PROGRAM ST5_MOTOR_1
VAR
	ClearFault: FB_ClearFault;
	SetEnableState: FB_SetEnableState;
	SetHomingParameter: FB_SetHomingParameter;
	FindHome: FB_FindHome;
	POSITION: DINT;
	GetMovementState: FB_GetMovementState;
	MoveToPosition: FB_MoveToPosition;
	SetOperationMode: FB_SetOperationMode;
	SetMotorParameter: FB_SetMotorParameter;
	SetPositionProfile: FB_SetPositionProfile;
END_VAR

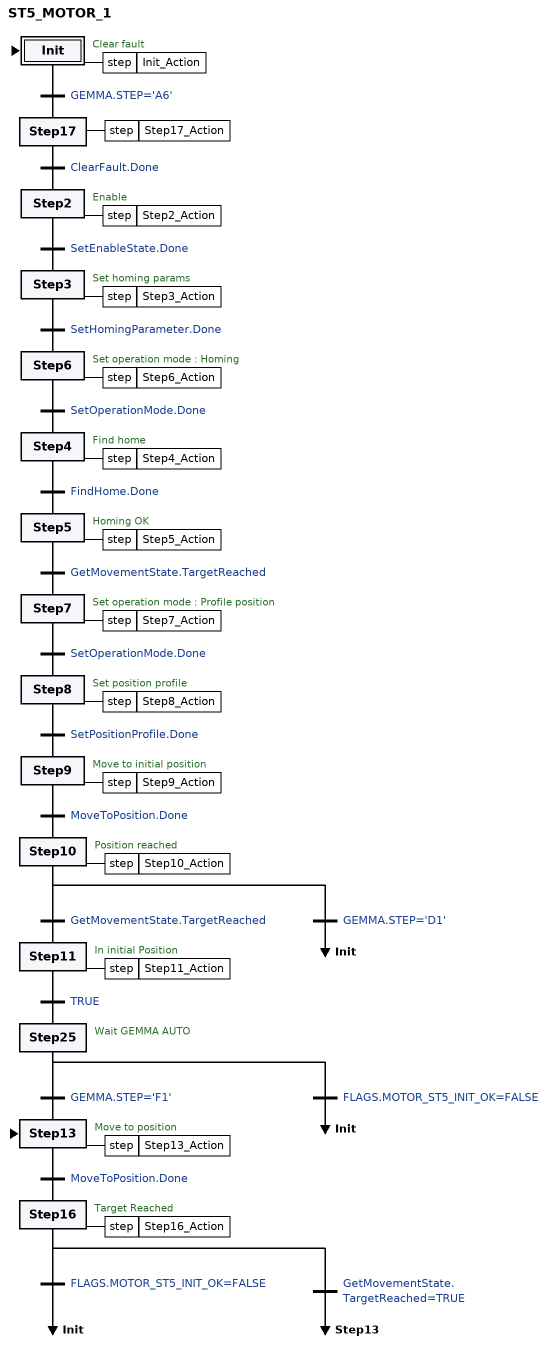
// Clear fault
INITIAL_STEP Init:
    Init_Action(N);  // step action
END_STEP
TRANSITION FROM Init TO Step17
    := GEMMA.STEP='A6';
END_TRANSITION
STEP Step17:
    Step17_Action(N);  // step action
END_STEP
TRANSITION FROM Step17 TO Step2
    := ClearFault.Done;
END_TRANSITION
// Enable
STEP Step2:
    Step2_Action(N);  // step action
END_STEP
TRANSITION FROM Step2 TO Step3
    := SetEnableState.Done;
END_TRANSITION
// Set homing params
STEP Step3:
    Step3_Action(N);  // step action
END_STEP
TRANSITION FROM Step3 TO Step6
    := SetHomingParameter.Done;
END_TRANSITION
// Set operation mode : Homing
STEP Step6:
    Step6_Action(N);  // step action
END_STEP
TRANSITION FROM Step6 TO Step4
    := SetOperationMode.Done;
END_TRANSITION
// Find home
STEP Step4:
    Step4_Action(N);  // step action
END_STEP
TRANSITION FROM Step4 TO Step5
    := FindHome.Done;
END_TRANSITION
// Homing OK
STEP Step5:
    Step5_Action(N);  // step action
END_STEP
TRANSITION FROM Step5 TO Step7
    := GetMovementState.TargetReached;
END_TRANSITION
// Set operation mode : Profile position
STEP Step7:
    Step7_Action(N);  // step action
END_STEP
TRANSITION FROM Step7 TO Step8
    := SetOperationMode.Done;
END_TRANSITION
// Set position profile
STEP Step8:
    Step8_Action(N);  // step action
END_STEP
TRANSITION FROM Step8 TO Step9
    := SetPositionProfile.Done;
END_TRANSITION
// Move to initial position
STEP Step9:
    Step9_Action(N);  // step action
END_STEP
TRANSITION FROM Step9 TO Step10
    := MoveToPosition.Done;
END_TRANSITION
// Position reached
STEP Step10:
    Step10_Action(N);  // step action
END_STEP
TRANSITION FROM Step10 TO Step11
    := GetMovementState.TargetReached;
END_TRANSITION
TRANSITION FROM Step10 TO Init
    := GEMMA.STEP='D1';
END_TRANSITION
// In initial Position
STEP Step11:
    Step11_Action(N);  // step action
END_STEP
TRANSITION FROM Step11 TO Step25
    := TRUE;
END_TRANSITION
// Wait GEMMA AUTO
STEP Step25:
END_STEP
TRANSITION FROM Step25 TO Step13
    := GEMMA.STEP='F1';
END_TRANSITION
TRANSITION FROM Step25 TO Init
    := FLAGS.MOTOR_ST5_INIT_OK=FALSE;
END_TRANSITION
// Move to position
STEP Step13:
    Step13_Action(N);  // step action
END_STEP
TRANSITION FROM Step13 TO Step16
    := MoveToPosition.Done;
END_TRANSITION
// Target Reached
STEP Step16:
    Step16_Action(N);  // step action
END_STEP
TRANSITION FROM Step16 TO Init
    := FLAGS.MOTOR_ST5_INIT_OK=FALSE;
END_TRANSITION
TRANSITION FROM Step16 TO Step13
    := GetMovementState.TargetReached=TRUE;
END_TRANSITION

ACTION Step6_Action:
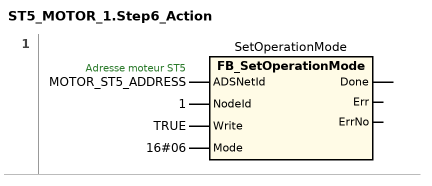
// NETWORK 1
//   MOTOR_ST5_ADDRESS: Adresse moteur ST5
SetOperationMode(ADSNetId := MOTOR_ST5_ADDRESS, NodeId := 1, Write := TRUE, Mode := 16#06); // FB_SetOperationMode
END_ACTION

ACTION Step2_Action:
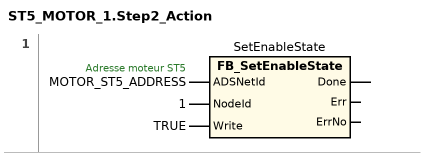
// NETWORK 1
//   MOTOR_ST5_ADDRESS: Adresse moteur ST5
SetEnableState(ADSNetId := MOTOR_ST5_ADDRESS, NodeId := 1, Write := TRUE); // FB_SetEnableState
END_ACTION

ACTION Step10_Action:
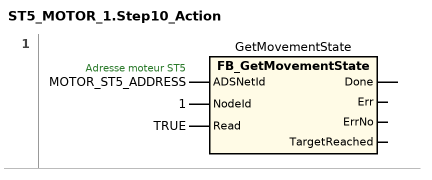
// NETWORK 1
//   MOTOR_ST5_ADDRESS: Adresse moteur ST5
GetMovementState(ADSNetId := MOTOR_ST5_ADDRESS, NodeId := 1, Read := TRUE); // FB_GetMovementState
END_ACTION

ACTION Step8_Action:
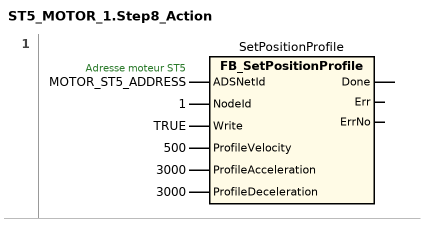
// NETWORK 1
//   MOTOR_ST5_ADDRESS: Adresse moteur ST5
SetPositionProfile(
    ADSNetId := MOTOR_ST5_ADDRESS,
    NodeId := 1,
    Write := TRUE,
    ProfileVelocity := 500,
    ProfileAcceleration := 3000,
    ProfileDeceleration := 3000); // FB_SetPositionProfile
END_ACTION

ACTION Step4_Action:
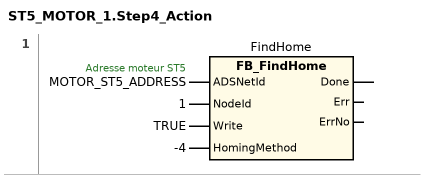
// NETWORK 1
//   MOTOR_ST5_ADDRESS: Adresse moteur ST5
FindHome(ADSNetId := MOTOR_ST5_ADDRESS, NodeId := 1, Write := TRUE, HomingMethod := -4); // FB_FindHome
END_ACTION

ACTION Step11_Action:

(*SetDisableState(
	ADSNetId:= '10.0.0.31.6.1',
	NodeId:= 1,
	Write:= TRUE);*)

FLAGS.MOTOR_ST5_INIT_OK:=TRUE;
END_ACTION

ACTION Step17_Action:
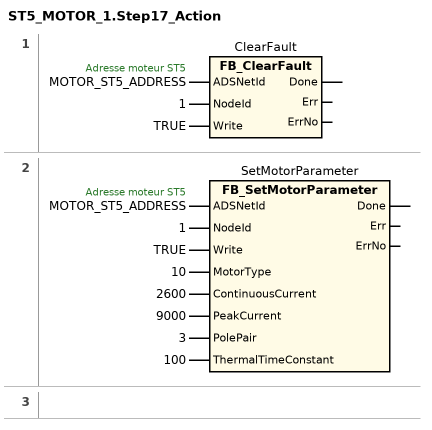
// NETWORK 1
//   MOTOR_ST5_ADDRESS: Adresse moteur ST5
ClearFault(ADSNetId := MOTOR_ST5_ADDRESS, NodeId := 1, Write := TRUE); // FB_ClearFault

// NETWORK 2
//   MOTOR_ST5_ADDRESS: Adresse moteur ST5
SetMotorParameter(
    ADSNetId := MOTOR_ST5_ADDRESS,
    NodeId := 1,
    Write := TRUE,
    MotorType := 10,
    ContinuousCurrent := 2600,
    PeakCurrent := 9000,
    PolePair := 3,
    ThermalTimeConstant := 100); // FB_SetMotorParameter

// NETWORK 3
END_ACTION

ACTION Step5_Action:
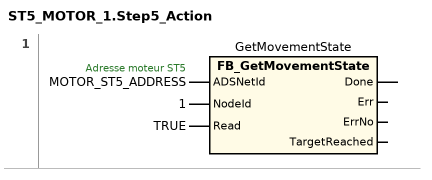
// NETWORK 1
//   MOTOR_ST5_ADDRESS: Adresse moteur ST5
GetMovementState(ADSNetId := MOTOR_ST5_ADDRESS, NodeId := 1, Read := TRUE); // FB_GetMovementState
END_ACTION

ACTION Step16_Action:
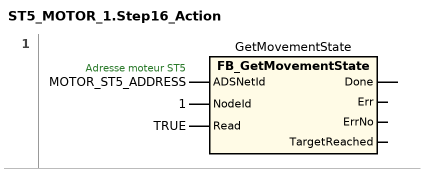
// NETWORK 1
//   MOTOR_ST5_ADDRESS: Adresse moteur ST5
GetMovementState(ADSNetId := MOTOR_ST5_ADDRESS, NodeId := 1, Read := TRUE); // FB_GetMovementState
END_ACTION

ACTION Init_Action:

END_ACTION

ACTION Step13_Action:
(*Limitation deplacement Moteur*)
IF FLAGS.MOTOR_ST5_POSITION>MOTOR_ST5_POSITION_MAX THEN
	POSITION:=MOTOR_ST5_POSITION_MAX;
ELSIF FLAGS.MOTOR_ST5_POSITION<0 THEN
	POSITION:=0;
ELSE
	POSITION:=FLAGS.MOTOR_ST5_POSITION;
END_IF


MoveToPosition(
	ADSNetId:= MOTOR_ST5_ADDRESS,
	NodeId:= 1,
	Write:= TRUE,
	TargetPosition:= POSITION,
	Absolut:= TRUE);
END_ACTION

ACTION Step3_Action:
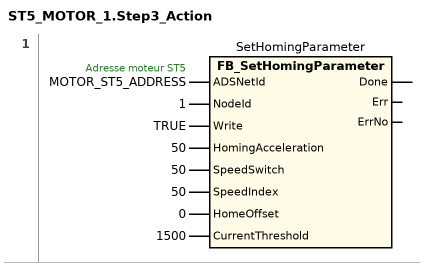
// NETWORK 1
//   MOTOR_ST5_ADDRESS: Adresse moteur ST5
SetHomingParameter(
    ADSNetId := MOTOR_ST5_ADDRESS,
    NodeId := 1,
    Write := TRUE,
    HomingAcceleration := 50,
    SpeedSwitch := 50,
    SpeedIndex := 50,
    HomeOffset := 0,
    CurrentThreshold := 1500); // FB_SetHomingParameter
END_ACTION

ACTION Step7_Action:
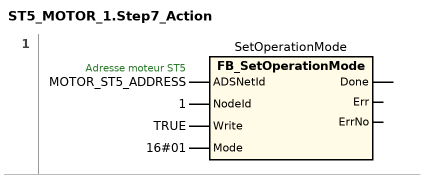
// NETWORK 1
//   MOTOR_ST5_ADDRESS: Adresse moteur ST5
SetOperationMode(ADSNetId := MOTOR_ST5_ADDRESS, NodeId := 1, Write := TRUE, Mode := 16#01); // FB_SetOperationMode
END_ACTION

ACTION Step9_Action:
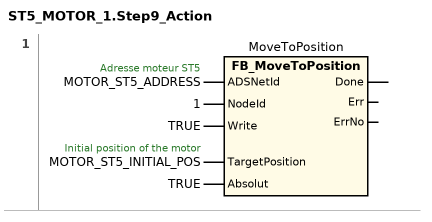
// NETWORK 1
//   MOTOR_ST5_ADDRESS: Adresse moteur ST5
//   MOTOR_ST5_INITIAL_POS: Initial position of the motor
MoveToPosition(
    ADSNetId := MOTOR_ST5_ADDRESS,
    NodeId := 1,
    Write := TRUE,
    TargetPosition := MOTOR_ST5_INITIAL_POS,
    Absolut := TRUE); // FB_MoveToPosition
END_ACTION

END_PROGRAM

(* stored: Version 1.1.0.1, ProductVersion 3.1.0.26
   POU ST5_MOTOR_1: Id {8a4ed119-4474-4692-b411-8c27cde9d7dd}
   Action Step6_Action: Id {0e4fd623-7450-4abb-b2d3-7cc16c9ed765}
   Action Step2_Action: Id {1076aeea-8a15-41e5-a210-6c86e040ef66}
   Action Step10_Action: Id {206bf2f5-c68b-403b-b9f9-9b59b3771269}
   Action Step8_Action: Id {3136b666-90bd-400e-b502-12d5b6e6cdc8}
   Action Step4_Action: Id {49cb329b-a749-4498-aca0-9cdec4278312}
   Action Step11_Action: Id {4f4d9624-02b8-4b16-883d-ade939c67cda}
   Action Step17_Action: Id {78a7b7c5-8261-4380-8a61-aeb89917e5c4}
   Action Step5_Action: Id {8c68eb7f-8030-4668-8377-9a5c9a1cf165}
   Action Step16_Action: Id {b62f7afa-bc32-465d-948c-da9e0687bece}
   Action Init_Action: Id {d0ee1788-2a7e-4f60-bdba-a5af602e9d8b}
   Action Step13_Action: Id {d8941ba6-6bee-470d-b335-cd62d727bbda}
   Action Step3_Action: Id {f14b4e47-77e2-451e-aad4-906f1aff2096}
   Action Step7_Action: Id {f523ea58-924b-417e-82b7-e18280964cd3}
   Action Step9_Action: Id {ffd3cc73-226e-42fa-baeb-9ec3e02f9a19} *)
